Fanuc KAREL source: bank_class.klc

PROGRAM class_name
%NOBUSYLAMP
%COMMENT = 'base bank class'
%NOLOCKGROUP
%UNINITVARS

%include namespace.m

CONST
  ER_WARN          = 0 -- warning no change in task execution
  ER_WARN_STP      = 1 -- pause all taks and stop all motion
  ER_ABORT         = 2 -- abort all tasks and cancel
  SUCCESS          = 0 -- success constant
  EXISTS           = 7015 -- Already exists code

VAR
  acc_number : INTEGER
  acc_name : STRING[32]
  acc_funds : REAL
  ledger : STRING[32]
  ledger_prog : STRING[32]

%include bank_class.klh
%from strings.klh %import i_to_s, r_to_s

-- hashstr
%class hashstr('hash.klc','hashclass.klh','hashstring.klt')


--error functions
ROUTINE CHK_STAT(rec_stat: INTEGER)
BEGIN
  IF(rec_stat <> SUCCESS) AND (rec_stat <> EXISTS) THEN
      POST_ERR(rec_stat,'',0, ER_ABORT)
  ENDIF
END CHK_STAT


ROUTINE karelError(errStr : STRING; errorType : INTEGER)
-- Error Type:
-- 0 : WARNING
-- 1 : WARNING + SHOWN IN HISTORY
-- 2 : ABORT
------------------------------------------
BEGIN
  CLR_IO_STAT(TPDISPLAY)
  WRITE TPDISPLAY(CR,CR, errStr)
  WRITE TPDISPLAY(CR,CR,CR,CR,CR,CR,CR,CR)
  FORCE_SPMENU(TP_PANEL, SPI_TPUSER, 1)
  POST_ERR(122043, '', 0 , errorType)
END karelError

--initialization
ROUTINE constructor
  VAR
    b : BOOLEAN
  BEGIN
    --set number
    acc_number = number
    --link account to ledger
    ledger = ldgr
    ledger_prog = ldgr_prog
    -- link account id to class_name
    b = hashstr__put(i_to_s(number), 'class_name', ldgr_prog, ldgr)
    IF NOT b THEN
      karelError('Issue in class_name writing to hash', ER_ABORT)
    ENDIF
  END constructor

ROUTINE desctructor
  VAR
    d_num : ARRAY[1] OF INTEGER
    d_nam : ARRAY[1] OF STRING[32]
    d_funds : ARRAY[1] OF REAL
    b : BOOLEAN
    e,s : INTEGER
  BEGIN
    --remove from ledger
    -- ** must do first as acc_number could be uninitialized
    b = hashstr__delete(i_to_s(acc_number), ledger_prog, ledger)
    IF NOT b THEN
      karelError('Issue removing '+ i_to_s(acc_number)+' from hash in class_name', ER_ABORT)
    ENDIF

    -- uninitialize class attributes
    SET_VAR(e,'class_name','acc_number',d_num[1],s)
    IF s=12311 THEN s= 0 ;ENDIF
    CHK_STAT(s)
    SET_VAR(e,'class_name','acc_name',d_nam[1],s)
    IF s=12311 THEN s= 0 ;ENDIF
    CHK_STAT(s)
    SET_VAR(e,'class_name','acc_funds',d_funds[1],s)
    IF s=12311 THEN s= 0 ;ENDIF
    CHK_STAT(s)
    SET_VAR(e,'class_name','ledger',d_nam[1],s)
    IF s=12311 THEN s= 0 ;ENDIF
    CHK_STAT(s)
    SET_VAR(e,'class_name','ledger_prog',d_nam[1],s)
    IF s=12311 THEN s= 0 ;ENDIF
    CHK_STAT(s)
  END desctructor

--getters

ROUTINE get_account_number
  BEGIN
    RETURN(acc_number)
  END get_account_number

ROUTINE get_account_name
  BEGIN
    RETURN(acc_name)
  END get_account_name

ROUTINE get_account_funds
  BEGIN
    RETURN(acc_funds)
  END get_account_funds

--setters

ROUTINE set_account_number
  VAR
    b : BOOLEAN
  BEGIN
    --delete previous ledger link
    b = hashstr__delete(i_to_s(acc_number), ledger_prog, ledger)
    IF NOT b THEN
      karelError('Issue removing '+ i_to_s(acc_number)+' from hash in class_name', ER_ABORT)
    ENDIF
    --set number
    acc_number = number
    --set new account number on ledger
    b = hashstr__put(i_to_s(number), 'class_name', ledger_prog, ledger)
    IF NOT b THEN
      karelError('Issue in class_name writing to hash', ER_ABORT)
    ENDIF
  END set_account_number

ROUTINE set_account_name
  BEGIN
    acc_name = name
  END set_account_name

ROUTINE set_account_funds
  BEGIN
    acc_funds = funds
  END set_account_funds

ROUTINE print_account
  BEGIN
    WRITE (CR,'id#', i_to_s(acc_number), ': ')
    WRITE (acc_name)
    WRITE (' Funds: $', r_to_s(acc_funds),CR)
  END print_account

ROUTINE transfer
  VAR
    new_bal : REAL
    prog_name : STRING[12]
    e,s : INTEGER
    b : BOOLEAN
  BEGIN
    -- set new balance for owner
    acc_funds = acc_funds - amount
    --get object of recipient
    b = hashstr__get(i_to_s(recipient), prog_name, ledger_prog, ledger)
    -- set new balance for recipient
    GET_VAR(e, prog_name, 'acc_funds', new_bal, s)
    CHK_STAT(s)
    new_bal = new_bal + amount
    SET_VAR(e, prog_name,'acc_funds',new_bal,s)
    CHK_STAT(s)

  END transfer

ROUTINE deposit
  BEGIN
    acc_funds = acc_funds + amount
  END deposit

BEGIN
END class_name
